// TIA Portal project "Assembler 1_Working_2_Only green" (V13)
// Vorlageprojekt für das Buch mit Zielsystem S7-1200

(* hardware
DEVICE "S7-1200-Station_1"  S7-1200 Station
   slot 0: "Baugruppenträger_0"  Rack  V1.0
   slot 1: "PLC_1"  CPU 1212C AC/DC/Rly  6ES7 212-1BE40-0XB0  V4.1
DEVICE "HMI_1"  KTP400 Basic PN
   slot 0: "HMI"  HMI  6AV2 123-2DB03-0AX0  13.0.1.0
   slot 1: "HMI_RT_1"  KTP400 Basic PN  6AV2 123-2DB03-0AX0  13.0.1.0
   slot 5: "HMI_1.IE_CP_1"  PROFINET Interface
      slot 1: "PROFINET Interface_1"  PROFINET Interface
         slot 1: "Port_1"  Port
*)

// ===== PLC "PLC_1"  CPU 1212C AC/DC/Rly =====

VAR_GLOBAL   // PLC tag table "Standard-Variablentabelle"
   "Moving x" AT %I0.0 : Bool;
   "Moving z" AT %I0.1 : Bool;
   "Iten detected" AT %I0.2 : Bool;
   "Lid at place" AT %I0.3 : Bool;
   "Lit Clamped" AT %I0.4 : Bool;
   "Pos at limit (lids)" AT %I0.5 : Bool;
   "Base at place" AT %I0.6 : Bool;
   "Base clamped" AT %I0.7 : Bool;
   "Pos at limit (base)" AT %I1.0 : Bool;
   "Part leaving" AT %I1.1 : Bool;
   "Start" AT %M100.0 : Bool;
   "Reset" AT %M100.1 : Bool;
   "Stop" AT %M100.2 : Bool;
   "E Stop" AT %M100.3 : Bool;
   "Move X" AT %Q0.0 : Bool;
   "Move z" AT %Q0.1 : Bool;
   "Grab" AT %Q0.2 : Bool;
   "Lids Conveyor" AT %Q0.3 : Bool;
   "Clamp Lid" AT %Q0.4 : Bool;
   "Pos raise (lids)" AT %Q0.5 : Bool;
   "Bases conveyor" AT %Q0.6 : Bool;
   "Clamp Base" AT %Q0.7 : Bool;
   "Pose Raise(base)" AT %Q1.0 : Bool;
   "Emitter 1" AT %Q1.1 : Bool;
   "Emitter 2" AT %Q1.2 : Bool;
   "Stop Light" AT %Q1.3 : Bool;
   "Green Objects" AT %QW30 : Word;
   "Tag_1" AT %M0.0 : Bool;
   "Tag_2" AT %M0.2 : Bool;
   "Tag_3" AT %M0.3 : Bool;
   "Tag_4" AT %M0.4 : Bool;
   "Tag_5" AT %M0.5 : Bool;
   "Tag_6" AT %M0.6 : Bool;
   "Tag_7" AT %M1.0 : Bool;
   "Tag_8" AT %M5.0 : Bool;
   "Tag_9" AT %M1.1 : Bool;
   "Tag_10" AT %M1.2 : Bool;
   "Tag_11" AT %M2.4 : Bool;
   "Tag_12" AT %M1.4 : Bool;
   "Tag_13" AT %M2.0 : Bool;
   "Tag_14" AT %M2.3 : Bool;
   "Tag_15" AT %M2.5 : Bool;
   "Tag_16" AT %M3.0 : Bool;
   "Tag_17" AT %M3.3 : Bool;
   "Tag_18" AT %M4.0 : Bool;
   "Start_Stop bit" AT %M5.5 : Bool;
   "Lid Color" AT %ID30 : DWord;
   "Lid" AT %M50.0 : Bool;
   "Base color" AT %ID34 : DWord;
   "Base" AT %M50.1 : Bool;
   "Rising edge Green lid" AT %M50.3 : Bool;
   "Rising edge Green base" AT %M50.4 : Bool;
   "Tag_19" AT %M6.0 : Bool;
   "Lid color input" AT %MB110 : Byte;
   "Base color input 1" AT %MB111 : Byte;
   "Base Color Input 2" AT %MB112 : Byte;
   "Green and Blue bit" AT %M50.5 : Bool;
   "Blue Objects" AT %QW34 : Word;
   "Base clamped FE" AT %M50.6 : Bool;
   "Base clamped FE2" AT %M50.7 : Bool;
END_VAR

// folder: System blocks/Program resources

DATA_BLOCK "IEC_Timer_0_DB"   // DB1
{ S7_Optimized_Access := 'FALSE' }
AUTHOR : Simatic
FAMILY : IEC
NAME : IEC_TMR
VERSION : 1.0
// stored: InstanceOfName ?
"?"
BEGIN
END_DATA_BLOCK

DATA_BLOCK "IEC_Timer_0_DB_1"   // DB2
{ S7_Optimized_Access := 'FALSE' }
AUTHOR : Simatic
FAMILY : IEC
NAME : IEC_TMR
VERSION : 1.0
// stored: InstanceOfName ?
"?"
BEGIN
END_DATA_BLOCK

DATA_BLOCK "IEC_Timer_0_DB_2"   // DB3
{ S7_Optimized_Access := 'FALSE' }
AUTHOR : Simatic
FAMILY : IEC
NAME : IEC_TMR
VERSION : 1.0
// stored: InstanceOfName ?
"?"
BEGIN
END_DATA_BLOCK

// folder: (top level)

FUNCTION "MHJ-PLC-Lab-Function-S71200" : Void   // FC9000, SCL
{ S7_Optimized_Access := 'FALSE' }
VERSION : 0.1
BEGIN

   #Value:=PEEK(area := 16#82,
        dbNumber := 0,
        byteOffset := 511);
   #Value := #Value + 1;

   POKE(area := 16#82,
        dbNumber := 0,
        byteOffset := 511,
        value := #Value);

   POKE(area:=16#81,
        dbNumber:=0,
        byteOffset:=1016,
        value:=#Value_01_DW);
   POKE(area := 16#81,
        dbNumber := 0,
        byteOffset := 1020,
        value := #Value_02_DW);

   POKE(area := 16#81,
        dbNumber := 0,
        byteOffset := 511,
        value := B#16#00);

   FOR #forVal := 0 TO 120 DO
       FOR #forVal_2:=0 TO 10 DO
           #rdTimeReturn:=RD_SYS_T(#outputTime);
           #rdTimeReturn := WR_SYS_T(#outputTime);
           #rdTimeReturn := RD_SYS_T(#outputTime);
           #rdTimeReturn := WR_SYS_T(#outputTime);
       END_FOR;
       #SyncVal:= PEEK(area := 16#81,
                      dbNumber := 0,
                      byteOffset := 511);
       IF #SyncVal = #CompVal THEN
          GOTO M_1;
       END_IF;
   END_FOR;
   RETURN;

   M_1:
   POKE(area := 16#81,
        dbNumber := 0,
        byteOffset := 511,
        value := B#16#0);
END_FUNCTION

ORGANIZATION_BLOCK "Main"   // OB1, LAD, ProgramCycle
TITLE = "Main Program Sweep (Cycle)"
{ S7_Optimized_Access := 'FALSE' }
VERSION : 0.1
   VAR_TEMP   // added for the SCL form of the ladder/FBD networks
      _w1 : Bool;
      _w2 : Bool;
      _w3 : Bool;
      _w4 : Bool;
      _w5 : Bool;
      _w6 : Bool;
      _w7 : Bool;
      _w8 : Bool;
   END_VAR
BEGIN

REGION Network 1: Connection block for PLCSIM communication - Don't delete this network! / FB to link Factory IO and Siemens TIA
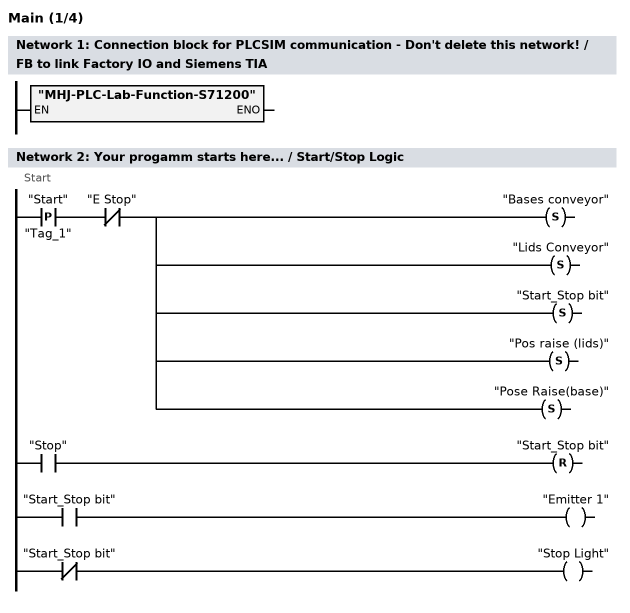
   RUNG wire#powerrail
      "MHJ-PLC-Lab-Function-S71200"()
   END_RUNG
   // the same network as SCL:
   "MHJ-PLC-Lab-Function-S71200"();
END_REGION

REGION Network 2: Your progamm starts here... / Start/Stop Logic
   // Start
   RUNG wire#powerrail
      P_Contact(operand := "Start", bit := "Tag_1")
      I_Contact( "E Stop" )
      wire#w1
      S_Coil( "Bases conveyor" )
   END_RUNG
   RUNG wire#w1
      S_Coil( "Lids Conveyor" )
   END_RUNG
   RUNG wire#w1
      S_Coil( "Start_Stop bit" )
   END_RUNG
   RUNG wire#w1
      S_Coil( "Pos raise (lids)" )
   END_RUNG
   RUNG wire#w1
      S_Coil( "Pose Raise(base)" )
   END_RUNG
   RUNG wire#powerrail
      Contact( "Stop" )
      R_Coil( "Start_Stop bit" )
   END_RUNG
   RUNG wire#powerrail
      Contact( "Start_Stop bit" )
      Coil( "Emitter 1" )
   END_RUNG
   RUNG wire#powerrail
      I_Contact( "Start_Stop bit" )
      Coil( "Stop Light" )
   END_RUNG
   // the same network as SCL:
   #_w1 := "Start" AND NOT "Tag_1";   // rising edge of "Start"
   "Tag_1" := "Start";
   IF #_w1 AND NOT "E Stop" THEN
       "Bases conveyor" := TRUE;
       "Lids Conveyor" := TRUE;
       "Start_Stop bit" := TRUE;
       "Pos raise (lids)" := TRUE;
       "Pose Raise(base)" := TRUE;
   END_IF;
   IF "Stop" THEN "Start_Stop bit" := FALSE; END_IF;
   "Emitter 1" := "Start_Stop bit";
   "Stop Light" := NOT "Start_Stop bit";
END_REGION

REGION Network 3: Step 1: Clamping the objects and bringing arm down - Based on color
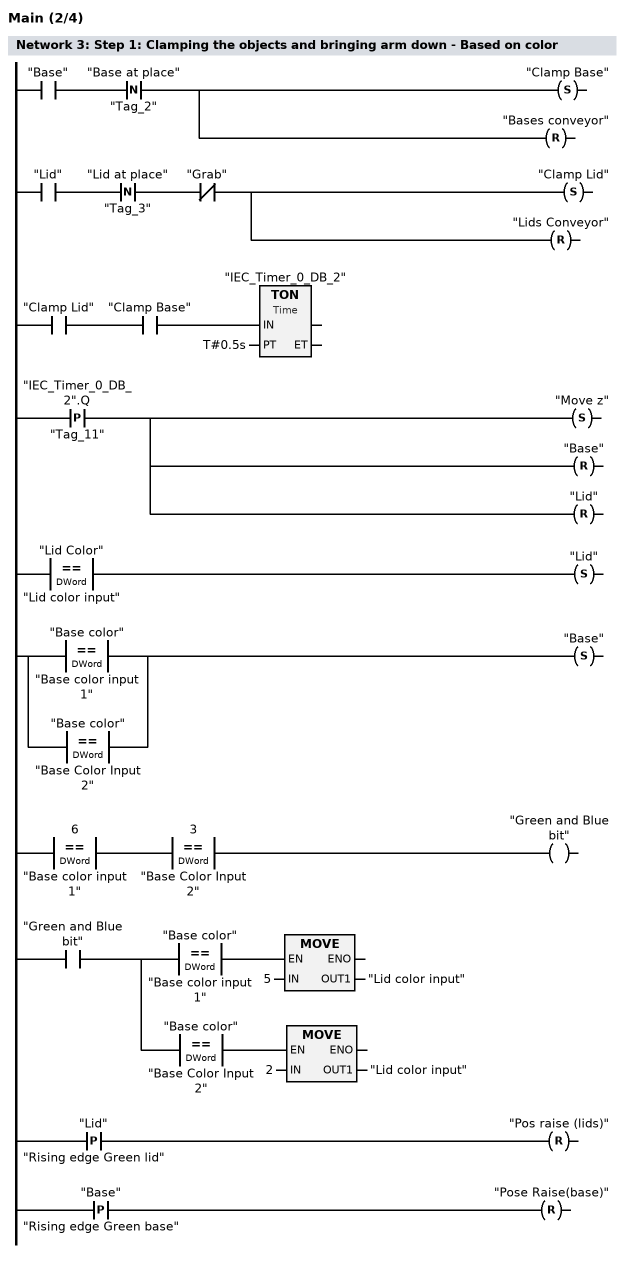
   #_w1 := "Base" AND NOT "Base at place" AND "Tag_2";   // falling edge of "Base at place"
   "Tag_2" := "Base at place";
   IF #_w1 THEN
       "Clamp Base" := TRUE;
       "Bases conveyor" := FALSE;
   END_IF;
   #_w2 := "Lid" AND NOT "Lid at place" AND "Tag_3";   // falling edge of "Lid at place"
   "Tag_3" := "Lid at place";
   IF #_w2 AND NOT "Grab" THEN
       "Clamp Lid" := TRUE;
       "Lids Conveyor" := FALSE;
   END_IF;
   "IEC_Timer_0_DB_2".TON(IN := "Clamp Lid" AND "Clamp Base", PT := T#0.5s);
   #_w3 := "IEC_Timer_0_DB_2".Q AND NOT "Tag_11";   // rising edge of "IEC_Timer_0_DB_2".Q
   "Tag_11" := "IEC_Timer_0_DB_2".Q;
   IF #_w3 THEN
       "Move z" := TRUE;
       "Base" := FALSE;
       "Lid" := FALSE;
   END_IF;
   IF "Lid Color" = "Lid color input" THEN "Lid" := TRUE; END_IF;
   IF ("Base color" = "Base color input 1") OR ("Base color" = "Base Color Input 2") THEN
       "Base" := TRUE;
   END_IF;
   "Green and Blue bit" := (6 = "Base color input 1") AND (3 = "Base Color Input 2");
   IF "Green and Blue bit" AND ("Base color" = "Base color input 1") THEN "Lid color input" := 5; END_IF;
   IF "Green and Blue bit" AND ("Base color" = "Base Color Input 2") THEN "Lid color input" := 2; END_IF;
   #_w4 := "Lid" AND NOT "Rising edge Green lid";   // rising edge of "Lid"
   "Rising edge Green lid" := "Lid";
   IF #_w4 THEN "Pos raise (lids)" := FALSE; END_IF;
   #_w5 := "Base" AND NOT "Rising edge Green base";   // rising edge of "Base"
   "Rising edge Green base" := "Base";
   IF #_w5 THEN "Pose Raise(base)" := FALSE; END_IF;
END_REGION

REGION Network 4: Picking the placing the object
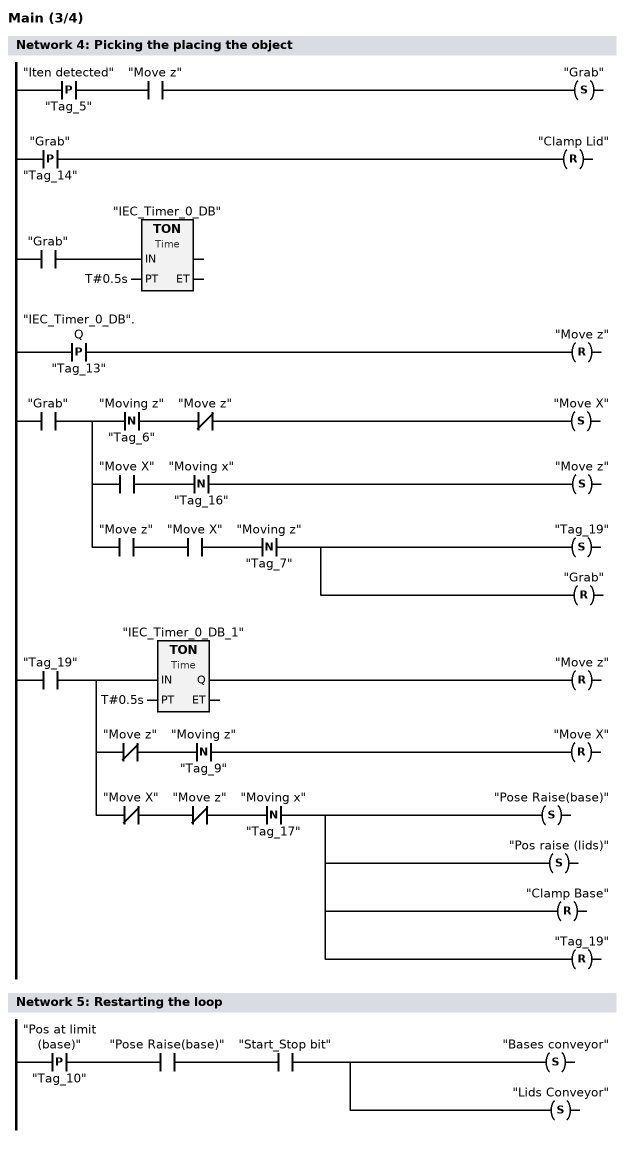
   #_w1 := "Iten detected" AND NOT "Tag_5";   // rising edge of "Iten detected"
   "Tag_5" := "Iten detected";
   IF #_w1 AND "Move z" THEN "Grab" := TRUE; END_IF;
   #_w2 := "Grab" AND NOT "Tag_14";   // rising edge of "Grab"
   "Tag_14" := "Grab";
   IF #_w2 THEN "Clamp Lid" := FALSE; END_IF;
   "IEC_Timer_0_DB".TON(IN := "Grab", PT := T#0.5s);
   #_w3 := "IEC_Timer_0_DB".Q AND NOT "Tag_13";   // rising edge of "IEC_Timer_0_DB".Q
   "Tag_13" := "IEC_Timer_0_DB".Q;
   IF #_w3 THEN "Move z" := FALSE; END_IF;
   #_w4 := "Grab" AND NOT "Moving z" AND "Tag_6";   // falling edge of "Moving z"
   "Tag_6" := "Moving z";
   IF #_w4 AND NOT "Move z" THEN "Move X" := TRUE; END_IF;
   #_w5 := "Grab" AND "Move X" AND NOT "Moving x" AND "Tag_16";   // falling edge of "Moving x"
   "Tag_16" := "Moving x";
   IF #_w5 THEN "Move z" := TRUE; END_IF;
   #_w6 := "Grab" AND "Move z" AND "Move X" AND NOT "Moving z" AND "Tag_7";   // falling edge of "Moving z"
   "Tag_7" := "Moving z";
   IF #_w6 THEN
       "Tag_19" := TRUE;
       "Grab" := FALSE;
   END_IF;
   "IEC_Timer_0_DB_1".TON(IN := "Tag_19", PT := T#0.5s);
   IF "IEC_Timer_0_DB_1".Q THEN "Move z" := FALSE; END_IF;
   #_w7 := "Tag_19" AND NOT "Move z" AND NOT "Moving z" AND "Tag_9";   // falling edge of "Moving z"
   "Tag_9" := "Moving z";
   IF #_w7 THEN "Move X" := FALSE; END_IF;
   #_w8 := "Tag_19" AND NOT "Move X" AND NOT "Move z" AND NOT "Moving x" AND "Tag_17";   // falling edge of "Moving x"
   "Tag_17" := "Moving x";
   IF #_w8 THEN
       "Pose Raise(base)" := TRUE;
       "Pos raise (lids)" := TRUE;
       "Clamp Base" := FALSE;
       "Tag_19" := FALSE;
   END_IF;
END_REGION

REGION Network 5: Restarting the loop
   RUNG wire#powerrail
      P_Contact(operand := "Pos at limit (base)", bit := "Tag_10")
      Contact( "Pose Raise(base)" )
      Contact( "Start_Stop bit" )
      wire#w1
      S_Coil( "Bases conveyor" )
   END_RUNG
   RUNG wire#w1
      S_Coil( "Lids Conveyor" )
   END_RUNG
   // the same network as SCL:
   #_w1 := "Pos at limit (base)" AND NOT "Tag_10";   // rising edge of "Pos at limit (base)"
   "Tag_10" := "Pos at limit (base)";
   IF #_w1 AND "Pose Raise(base)" AND "Start_Stop bit" THEN
       "Bases conveyor" := TRUE;
       "Lids Conveyor" := TRUE;
   END_IF;
END_REGION

REGION Network 6: Emergency Stop condition
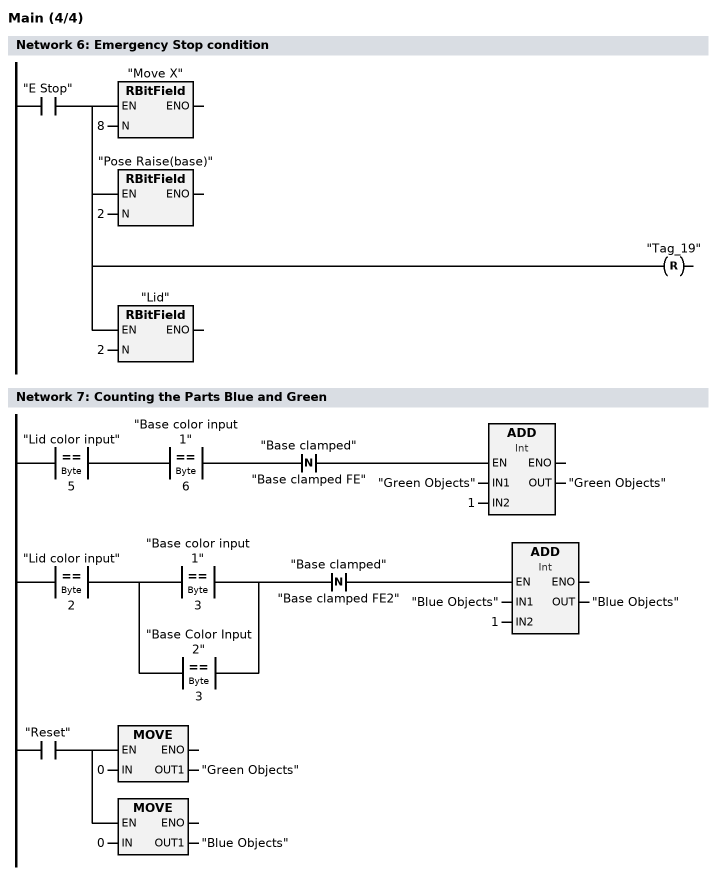
   // no SCL statement known for RBitField: written as a call
   #_w1 := "E Stop";
   IF #_w1 THEN
       RBitField(n := 8, operand := "Move X");
       RBitField(n := 2, operand := "Pose Raise(base)");
       "Tag_19" := FALSE;
       RBitField(n := 2, operand := "Lid");
   END_IF;
END_REGION

REGION Network 7: Counting the Parts Blue and Green
   RUNG wire#powerrail
      { S7_Templates := "SrcType := Byte" } EQ_Contact(in1 := "Lid color input", in2 := 5)
      { S7_Templates := "SrcType := Byte" } EQ_Contact(in1 := "Base color input 1", in2 := 6)
      N_Contact(operand := "Base clamped", bit := "Base clamped FE")
      { S7_Templates := "SrcType := Int"; S7_GenerateENO := "TRUE" } Add(in1 := "Green Objects", in2 := 1, out => "Green Objects")
   END_RUNG
   RUNG wire#powerrail
      { S7_Templates := "SrcType := Byte" } EQ_Contact(in1 := "Lid color input", in2 := 2)
      wire#w1
      { S7_Templates := "SrcType := Byte" } EQ_Contact(in1 := "Base color input 1", in2 := 3)
      wire#w2
      N_Contact(operand := "Base clamped", bit := "Base clamped FE2")
      { S7_Templates := "SrcType := Int"; S7_GenerateENO := "TRUE" } Add(in1 := "Blue Objects", in2 := 1, out => "Blue Objects")
   END_RUNG
   RUNG wire#w1
      { S7_Templates := "SrcType := Byte" } EQ_Contact(in1 := "Base Color Input 2", in2 := 3)
   END_RUNG wire#w2
   RUNG wire#powerrail
      Contact( "Reset" )
      wire#w3
      { S7_GenerateENO := "TRUE" } Move(in := 0, out1 => "Green Objects")
   END_RUNG
   RUNG wire#w3
      { S7_GenerateENO := "TRUE" } Move(in := 0, out1 => "Blue Objects")
   END_RUNG
   // the same network as SCL:
   #_w1 := ("Lid color input" = 5) AND ("Base color input 1" = 6) AND NOT "Base clamped" AND "Base clamped FE";   // falling edge of "Base clamped"
   "Base clamped FE" := "Base clamped";
   IF #_w1 THEN "Green Objects" := "Green Objects" + 1; END_IF;
   #_w2 := ("Lid color input" = 2) AND (("Base color input 1" = 3) OR ("Base Color Input 2" = 3)) AND NOT "Base clamped" AND "Base clamped FE2";   // falling edge of "Base clamped"
   "Base clamped FE2" := "Base clamped";
   IF #_w2 THEN "Blue Objects" := "Blue Objects" + 1; END_IF;
   IF "Reset" THEN
       "Green Objects" := 0;
       "Blue Objects" := 0;
   END_IF;
END_REGION
END_ORGANIZATION_BLOCK

(* ===== HMI "HMI_RT_1" =====
connection "HMI_Connection_1": ETHERNET, SMART_S7_1200_OMS

HMI tags "Default tag table"
   "Start" : Bool = PLC "Start", 1 s
   "Stop" : Bool = PLC "Stop", 1 s
   "E Stop" : Bool = PLC "E Stop", 1 s
   "Counter" : Word = PLC "Green Objects", 1 s
   "Lid color input" : Byte = PLC "Lid color input", 1 s
   "Base color input" : Byte = PLC "Base color input 1", 1 s
   "Base Color Input 2" : Byte = PLC "Base Color Input 2", 1 s
   "Green HMI" : Bool, internal
   "Blue HMI" : Bool, internal
   "GB1" : Bool, internal
   "GB2" : Bool, internal
   "Blue Objects" : Word = PLC "Blue Objects", 1 s
   "Reset" : Bool = PLC "Reset", 1 s

recipe "Color": Lid <- "Lid color input", Base 1 <- "Base color input", Base 2 <- "Base Color Input 2"

Template "Template_1" 480x272
   Button "Template_Button" at 388,227 size 63x44
   Button "Template_Button_1" at 268,227 size 63x44
   Button "Template_Button_2" at 148,227 size 63x44
   Button "Template_Button_3" at 28,227 size 63x44

screen "Root screen" 480x272, template "Template_1"
   Button "Button_1" at 27,68 size 96x32
   Button "Button_2" at 141,69 size 96x32
   Switch "Switch_1" at 25,126 size 142x32
   TextField "Text field_1" at 25,104 size 142x22
   IOField "I/O field_1" at 58,184 size 54x32
   TextField "Text field_2" at 20,164 size 74x20
   Button "Button_3" at 294,101 size 96x32
   Button "Button_4" at 294,141 size 96x32
   Button "Button_5" at 294,182 size 126x32
   IOField "I/O field_2" at 155,183 size 58x32
   TextField "Text field_3" at 118,164 size 85x20
   TextField "Text field_4" at 294,73 size 107x22
   TextField "Text field_5" at 22,42 size 139x22
   TextField "Text field_6" at 294,42 size 171x18
   TextField "Text field_7" at 294,57 size 149x18
   TextField "Text field_8" at 24,11 size 157x25
   TextField "Text field_9" at 294,20 size 80x22
   Button "Button_7" at 221,184 size 52x32
*)